TYPE ST_ITC_MCR :
(**************************************************************************************
 * 	Application		:	BoxControl Framework
 *	Revision		:	$Revision: 404529 $
 *	Revision date	:	$Date: 2018-04-23 08:21:38 +0200 (Mo., 23 Apr 2018) $
 *	Last changed by	:	$Author: b7bolm $
 *	URL				:	$URL: http://almscdc.swisslog.com/repo/SWPD/Development/BoxControlFramework/20_Release/trunk/01_Software/BCF/BCF/JumpStart/20_Product/10_App/11_Com/10_Lib/10_Conv/11_ITC/01_DUTs/ST_ITC_MCR.TcDUT $
 *
 *	Purpose			:	MCR Structure
 *
 * ------------------------------------------------------------------------------------
 *	Copyright Swisslog [IP AG], Switzerland. All rights reserved.
 * 
 * ------------------------------------------------------------------------------------
 *	
 * 	Revision History: 
 *
 * 	VERSION			DATE			INITIALS			DESCRIPTION
 *	0.1				01.01.2001		swl					Example
 *
 **************************************************************************************)
STRUCT
	Position			: STRING(Conveyor.POSITION_STRINGLENGTH); // 12 Digit SIS Location MM-GGG-EEEE-FF-Z 
	Code				: INT; // Code
	Mode				: INT; // Mode
	Speed				: ST_ITC_ManualMotionSpeed; // Speed
	Axis				: ARRAY[1..6] OF ST_ITC_ManualMotionAxis; // Axis
	Button				: ARRAY[1..2] OF ST_ITC_ManualMotionSelection; // Buttons
	eReturnCode			: E_ErrorConv; // Return code
END_STRUCT
END_TYPE

(* stored: Version 1.1.0.1, ProductVersion 3.1.4022.12
   DUT ST_ITC_MCR: Id {40e67d3a-3f6a-4fcb-8f39-e31bbc79ec99} *)
